# EPICS substitutions: kstar/siteApp/RBA/tags/20120203-LabVIEW-version/RBAApp/Db/userHost.substitutions
# Example substitutions file

file "db/dbExample1.db" {
    { user = "RBA" }
}

file db/dbExample2.db {
    pattern { user, no, scan }
        { "RBA", 1, "1 second" }
        { "RBA", 2, "2 second" }
        { "RBA", 3, "5 second" }
}
